{attribute 'GeneratedUsingTerminal: AMI8000-0000-0016'}
{attribute addProperty BoxType "AMI8000-0000-0016"}
{attribute addProperty Id "Target_positionAT %Q*UDINT4"}
{attribute addProperty CRC "86249236"}
{attribute addProperty Size "4"}
TYPE DRV_Target_position_05240F14 EXTENDS OutputBase_10CEE7DE :
STRUCT
	{attribute addProperty Name "Target_position"}
	Target_position AT %Q* : UDINT;
END_STRUCT
END_TYPE

(* stored: Version 1.2.0.0, ProductVersion 3.1.4024.11
   DUT DRV_Target_position_05240F14: Id {3efb771e-552a-4669-b1c7-5099d00c5ef1} *)
